TYPE E_UnistatState :
(
	Error := -1,
	Off := 0,
	On := 1
)DINT;
END_TYPE

(* stored: Version 1.1.0.1, ProductVersion 3.1.4024.6
   DUT E_UnistatState: Id {3edea4a5-59d2-4a13-a2a2-c7486155c3c6} *)
